Staubli VAL3: Form_LabelList.pgx

public program Form_LabelList(string x_sTitle, string x_sLabel, string& x_sLableList[], string x_sPanelTitle, string& x_sList[], num& x_nSelectIndex, string x_sBottom)
  local num l_nNum
begin

cls()
title(x_sTitle)
call Control_PanelXY(2,0,15,10)
call Control_Panel(x_sLabel)
for l_nNum=0 to size(x_sLableList)-1
  gotoxy(nPanelLTopX+1,nPanelLTopY+l_nNum+1)
  put(x_sLableList[l_nNum])
endFor

call Control_PanelXY(22,0,15,10)
call Control_Panel(x_sPanelTitle)
call Control_BottomS(x_sBottom)

//x_nSelectIndex=0
call Control_List(x_sList,x_nSelectIndex)



end
